{attribute 'qualified_only'}
VAR_GLOBAL CONSTANT PERSISTENT
	AXIS_FILTER_WHEEL : STRING := '1';
	
	// FILTER WHEEL
	FW_DRIVING_CURRENT_IN_PERCENT : UINT := 90;
	FW_HOLDING_CURRENT_IN_PERCENT : UINT := 50;
	FW_LIMIT_SWITCH_MASK : UINT := 0;
END_VAR

(* stored: Version 1.1.0.1, ProductVersion 3.1.4024.12
   GVL AxesConst: Id {1ae4207d-b739-435f-81db-02b6f0ac9386} *)
